Fanuc TP program (LS listing): m1_chuck_opn.ls

/PROG  M1_CHUCK_OPN
/ATTR
OWNER		= MNEDITOR;
COMMENT		= "";
PROG_SIZE	= 394;
CREATE		= DATE 19-04-08  TIME 11:32:36;
MODIFIED	= DATE 19-04-15  TIME 12:41:26;
FILE_NAME	= W1_CHUCK;
VERSION		= 0;
LINE_COUNT	= 14;
MEMORY_SIZE	= 874;
PROTECT		= READ_WRITE;
TCD:  STACK_SIZE	= 0,
      TASK_PRIORITY	= 50,
      TIME_SLICE	= 0,
      BUSY_LAMP_OFF	= 0,
      ABORT_REQUEST	= 0,
      PAUSE_REQUEST	= 0;
DEFAULT_GROUP	= 1,*,*,*,*;
CONTROL_CODE	= 00000000 00000000;
/APPL
/MN
   1:  DO[41:W1_CHUCK_OPEN]=PULSE,1.0sec ;
   2:  WAIT   3.00(sec) ;
   3:   ;
   4:  $WAITTMOUT=200 ;
   5:  WAIT (DI[49:W1_CHUCK_OPENED]) TIMEOUT,LBL[1] ;
   6:   ;
   7:   ;
   8:  END ;
   9:  LBL[1] ;
  10:  MESSAGE[...] ;
  11:  MESSAGE[PRIHVATNICA STROJA 1] ;
  12:  MESSAGE[NIJE OTVORILA] ;
  13:  WAIT (DI[49:W1_CHUCK_OPENED])    ;
  14:  END ;
/POS
/END
